// TwinCAT 3 PLC project BscNoComp
// ProgramVersion: 3.1.4026.13
// libraries:
//   CmpBitmapPool, * (System)
//   Tc2_Standard, * (Beckhoff Automation GmbH)
//   Tc2_System, * (Beckhoff Automation GmbH)
//   Tc3_Module, * (Beckhoff Automation GmbH)
//   VisuSymbols,3.5.10.0,System
// project tree:
//   GVLs/ G_Enables.TcGVL, G_FilterConstants.TcGVL, G_Mode.TcGVL (not stored), G_OPC.TcGVL, G_Parameters.TcGVL (not stored)
//   Input/ G_Input.TcGVL (not stored)
//   Output/ G_Output.TcGVL (not stored)
//   / PlcTask.TcTTO, Visualization Manager.TcVMO (not stored)
//   Program/ MAIN.TcPOU (not stored)
//   XML/ FB_Derivator.TcPOU (not stored), FB_Integrator.TcPOU (not stored), G_Init.TcGVL (not stored)

CONFIGURATION BscNoComp
    RESOURCE PLC ON TwinCAT3
        TASK PlcTask(INTERVAL := T#1ms, PRIORITY := 20);
    END_RESOURCE
END_CONFIGURATION

// ---- GVLs/G_Enables.TcGVL
{attribute 'qualified_only'}
VAR_GLOBAL
END_VAR

// ---- GVLs/G_FilterConstants.TcGVL
{attribute 'qualified_only'}
VAR_GLOBAL
END_VAR

// ---- GVLs/G_OPC.TcGVL
{attribute 'qualified_only'}
VAR_GLOBAL
END_VAR
